# EPICS autosave request: pmac/qcm_settings.req
$(P):ENERGYMODE
